// TIA Portal V16 export
// export: Created 2022-03-28T07:44:05.4925085Z, ExportSetting WithDefaults, DisplayName Totally Integrated Automation Portal, DisplayVersion V16 Update 5, DisplayName TIA Portal Version Control Interface, DisplayVersion V16 Update 2, DisplayName TIA Portal Openness, DisplayVersion V16 Update 5, DisplayName STEP 7 Professional, DisplayVersion V16 Update 5, DisplayName STEP 7 Safety, DisplayVersion V16, DisplayName WinCC Professional, DisplayVersion V16 Update 5
FUNCTION "fc_03_Alarms" : Void   // FC3, LAD
{ S7_Optimized_Access := 'TRUE' }
VERSION : 0.1
// stored: AutoNumber false, IsIECCheckEnabled false, SetENOAutomatically false, UDAEnableTagReadback false
   VAR_TEMP   // added for the SCL form of the ladder/FBD networks
      _w1 : Bool;
      _w2 : Bool;
      _w3 : Bool;
   END_VAR
BEGIN

REGION Network 1
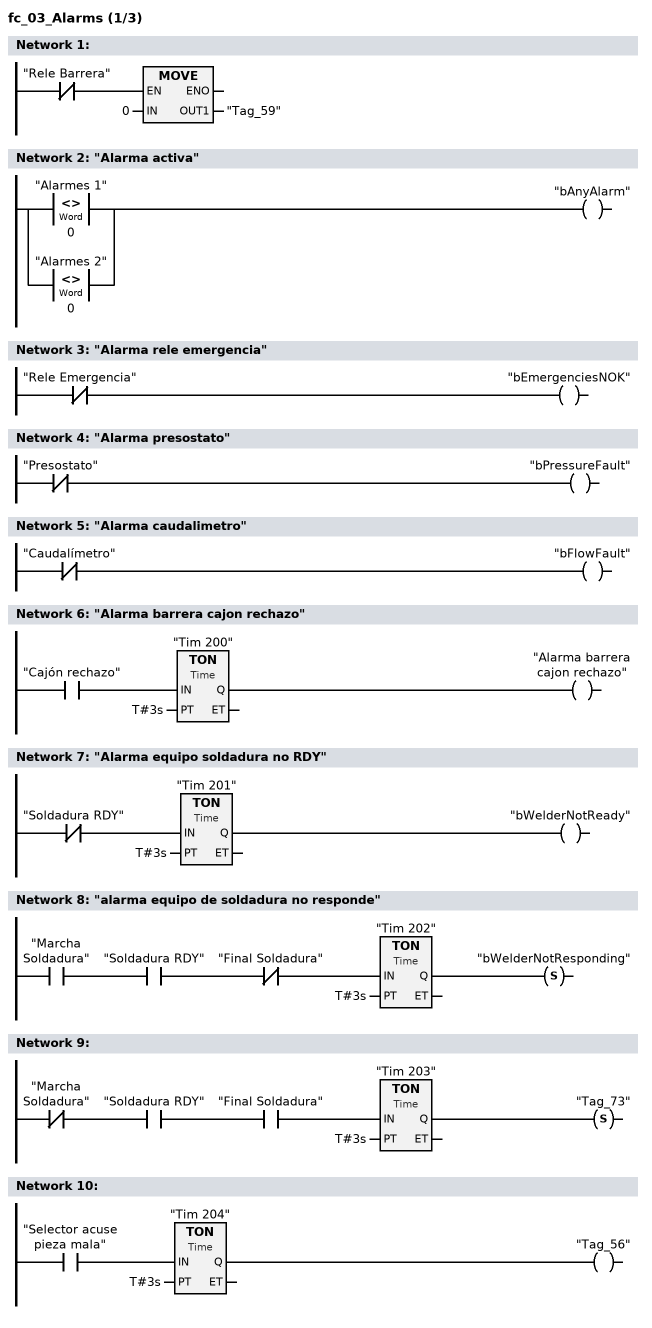
   RUNG wire#powerrail
      I_Contact( "Rele Barrera" )
      Move(in := 0, out1 => "Tag_59")
   END_RUNG
   // the same network as SCL:
   IF NOT "Rele Barrera" THEN "Tag_59" := 0; END_IF;
END_REGION

REGION Network 2: "Alarma activa"
   RUNG wire#powerrail
      { S7_Templates := "SrcType := Word" } NE_Contact(in1 := "Alarmes 1", in2 := 0)
      wire#w1
      Coil( "bAnyAlarm" )
   END_RUNG
   RUNG wire#powerrail
      { S7_Templates := "SrcType := Word" } NE_Contact(in1 := "Alarmes 2", in2 := 0)
   END_RUNG wire#w1
   // the same network as SCL:
   "bAnyAlarm" := ("Alarmes 1" <> 0) OR ("Alarmes 2" <> 0);
END_REGION

REGION Network 3: "Alarma rele emergencia"
   RUNG wire#powerrail
      I_Contact( "Rele Emergencia" )
      Coil( "bEmergenciesNOK" )
   END_RUNG
   // the same network as SCL:
   "bEmergenciesNOK" := NOT "Rele Emergencia";
END_REGION

REGION Network 4: "Alarma presostato"
   RUNG wire#powerrail
      I_Contact( "Presostato" )
      Coil( "bPressureFault" )
   END_RUNG
   // the same network as SCL:
   "bPressureFault" := NOT "Presostato";
END_REGION

REGION Network 5: "Alarma caudalimetro"
   RUNG wire#powerrail
      I_Contact( "Caudalímetro" )
      Coil( "bFlowFault" )
   END_RUNG
   // the same network as SCL:
   "bFlowFault" := NOT "Caudalímetro";
END_REGION

REGION Network 6: "Alarma barrera cajon rechazo"
   RUNG wire#powerrail
      Contact( "Cajón rechazo" )
      { S7_Templates := "time_type := Time" } "Tim 200".TON(pt := T#3s, et =>)
      Coil( "Alarma barrera cajon rechazo" )
   END_RUNG
   // the same network as SCL:
   "Tim 200".TON(IN := "Cajón rechazo", PT := T#3s);
   "Alarma barrera cajon rechazo" := "Tim 200".Q;
END_REGION

REGION Network 7: "Alarma equipo soldadura no RDY"
   RUNG wire#powerrail
      I_Contact( "Soldadura RDY" )
      { S7_Templates := "time_type := Time" } "Tim 201".TON(pt := T#3s, et =>)
      Coil( "bWelderNotReady" )
   END_RUNG
   // the same network as SCL:
   "Tim 201".TON(IN := NOT "Soldadura RDY", PT := T#3s);
   "bWelderNotReady" := "Tim 201".Q;
END_REGION

REGION Network 8: "alarma equipo de soldadura no responde"
   RUNG wire#powerrail
      Contact( "Marcha Soldadura" )
      Contact( "Soldadura RDY" )
      I_Contact( "Final Soldadura" )
      { S7_Templates := "time_type := Time" } "Tim 202".TON(pt := T#3s, et =>)
      S_Coil( "bWelderNotResponding" )
   END_RUNG
   // the same network as SCL:
   "Tim 202".TON(IN := "Marcha Soldadura" AND "Soldadura RDY" AND NOT "Final Soldadura", PT := T#3s);
   IF "Tim 202".Q THEN "bWelderNotResponding" := TRUE; END_IF;
END_REGION

REGION Network 9
   RUNG wire#powerrail
      I_Contact( "Marcha Soldadura" )
      Contact( "Soldadura RDY" )
      Contact( "Final Soldadura" )
      { S7_Templates := "time_type := Time" } "Tim 203".TON(pt := T#3s, et =>)
      S_Coil( "Tag_73" )
   END_RUNG
   // the same network as SCL:
   "Tim 203".TON(IN := NOT "Marcha Soldadura" AND "Soldadura RDY" AND "Final Soldadura", PT := T#3s);
   IF "Tim 203".Q THEN "Tag_73" := TRUE; END_IF;
END_REGION

REGION Network 10
   RUNG wire#powerrail
      Contact( "Selector acuse pieza mala" )
      { S7_Templates := "time_type := Time" } "Tim 204".TON(pt := T#3s, et =>)
      Coil( "Tag_56" )
   END_RUNG
   // the same network as SCL:
   "Tim 204".TON(IN := "Selector acuse pieza mala", PT := T#3s);
   "Tag_56" := "Tim 204".Q;
END_REGION

REGION Network 12: Alarmas Pinza 1
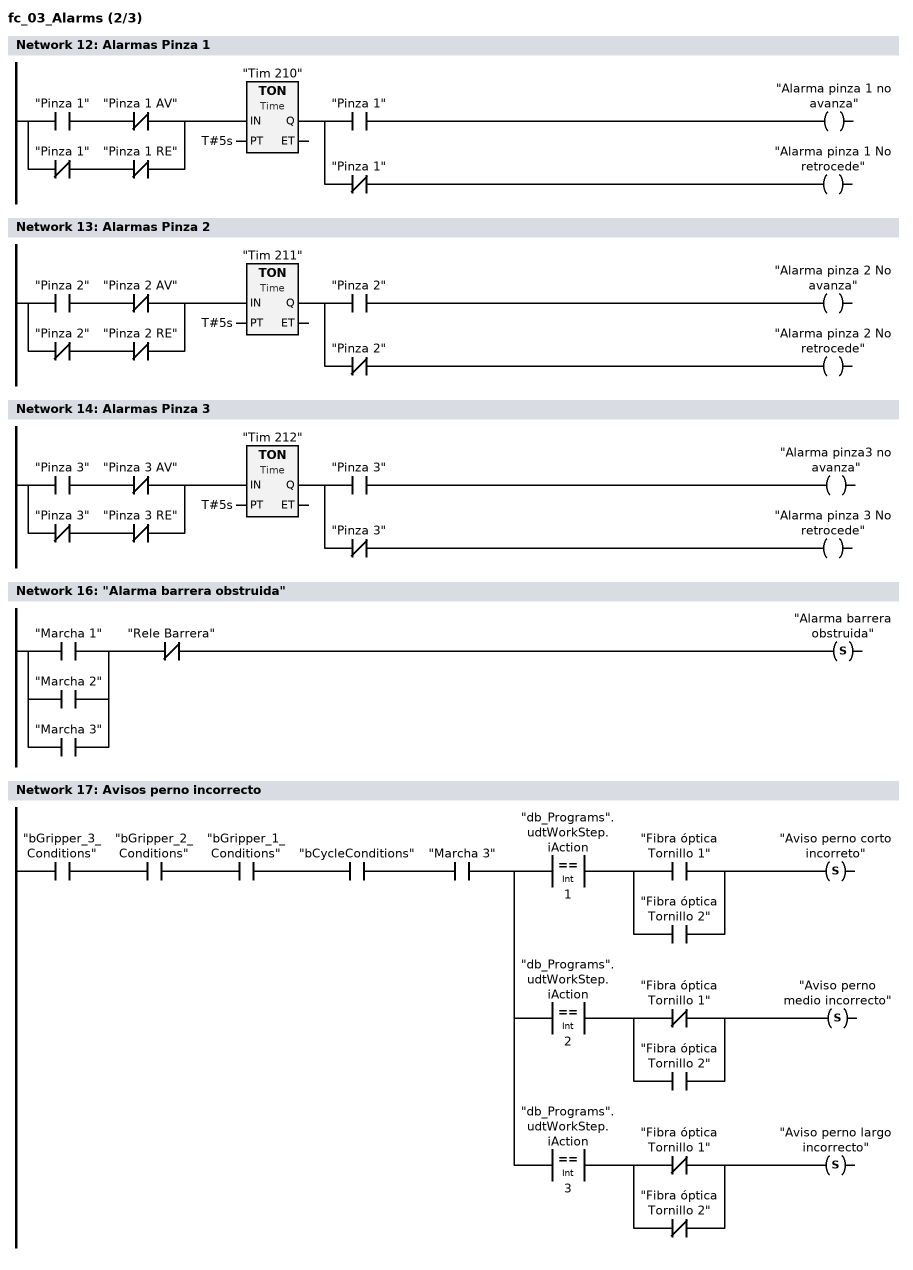
   RUNG wire#powerrail
      Contact( "Pinza 1" )
      I_Contact( "Pinza 1 AV" )
      wire#w1
      { S7_Templates := "time_type := Time" } "Tim 210".TON(pt := T#5s, et =>)
      wire#w2
      Contact( "Pinza 1" )
      Coil( "Alarma pinza 1 no avanza" )
   END_RUNG
   RUNG wire#powerrail
      I_Contact( "Pinza 1" )
      I_Contact( "Pinza 1 RE" )
   END_RUNG wire#w1
   RUNG wire#w2
      I_Contact( "Pinza 1" )
      Coil( "Alarma pinza 1 No retrocede" )
   END_RUNG
   // the same network as SCL:
   "Tim 210".TON(IN := ("Pinza 1" AND NOT "Pinza 1 AV") OR (NOT "Pinza 1" AND NOT "Pinza 1 RE"), PT := T#5s);
   "Alarma pinza 1 no avanza" := "Tim 210".Q AND "Pinza 1";
   "Alarma pinza 1 No retrocede" := "Tim 210".Q AND NOT "Pinza 1";
END_REGION

REGION Network 13: Alarmas Pinza 2
   RUNG wire#powerrail
      Contact( "Pinza 2" )
      I_Contact( "Pinza 2 AV" )
      wire#w1
      { S7_Templates := "time_type := Time" } "Tim 211".TON(pt := T#5s, et =>)
      wire#w2
      Contact( "Pinza 2" )
      Coil( "Alarma pinza 2 No avanza" )
   END_RUNG
   RUNG wire#powerrail
      I_Contact( "Pinza 2" )
      I_Contact( "Pinza 2 RE" )
   END_RUNG wire#w1
   RUNG wire#w2
      I_Contact( "Pinza 2" )
      Coil( "Alarma pinza 2 No retrocede" )
   END_RUNG
   // the same network as SCL:
   "Tim 211".TON(IN := ("Pinza 2" AND NOT "Pinza 2 AV") OR (NOT "Pinza 2" AND NOT "Pinza 2 RE"), PT := T#5s);
   "Alarma pinza 2 No avanza" := "Tim 211".Q AND "Pinza 2";
   "Alarma pinza 2 No retrocede" := "Tim 211".Q AND NOT "Pinza 2";
END_REGION

REGION Network 14: Alarmas Pinza 3
   RUNG wire#powerrail
      Contact( "Pinza 3" )
      I_Contact( "Pinza 3 AV" )
      wire#w1
      { S7_Templates := "time_type := Time" } "Tim 212".TON(pt := T#5s, et =>)
      wire#w2
      Contact( "Pinza 3" )
      Coil( "Alarma pinza3 no avanza" )
   END_RUNG
   RUNG wire#powerrail
      I_Contact( "Pinza 3" )
      I_Contact( "Pinza 3 RE" )
   END_RUNG wire#w1
   RUNG wire#w2
      I_Contact( "Pinza 3" )
      Coil( "Alarma pinza 3 No retrocede" )
   END_RUNG
   // the same network as SCL:
   "Tim 212".TON(IN := ("Pinza 3" AND NOT "Pinza 3 AV") OR (NOT "Pinza 3" AND NOT "Pinza 3 RE"), PT := T#5s);
   "Alarma pinza3 no avanza" := "Tim 212".Q AND "Pinza 3";
   "Alarma pinza 3 No retrocede" := "Tim 212".Q AND NOT "Pinza 3";
END_REGION

REGION Network 16: "Alarma barrera obstruida"
   RUNG wire#powerrail
      Contact( "Marcha 1" )
      wire#w1
      I_Contact( "Rele Barrera" )
      S_Coil( "Alarma barrera obstruida" )
   END_RUNG
   RUNG wire#powerrail
      Contact( "Marcha 2" )
   END_RUNG wire#w1
   RUNG wire#powerrail
      Contact( "Marcha 3" )
   END_RUNG wire#w1
   // the same network as SCL:
   IF ("Marcha 1" OR "Marcha 2" OR "Marcha 3") AND NOT "Rele Barrera" THEN
       "Alarma barrera obstruida" := TRUE;
   END_IF;
END_REGION

REGION Network 17: Avisos perno incorrecto
   RUNG wire#powerrail
      Contact( "bGripper_3_Conditions" )
      Contact( "bGripper_2_Conditions" )
      Contact( "bGripper_1_Conditions" )
      Contact( "bCycleConditions" )
      Contact( "Marcha 3" )
      wire#w1
      { S7_Templates := "SrcType := Int" } EQ_Contact(in1 := "db_Programs".udtWorkStep.iAction, in2 := 1)
      wire#w2
      Contact( "Fibra óptica Tornillo 1" )
      wire#w3
      S_Coil( "Aviso perno corto incorreto" )
   END_RUNG
   RUNG wire#w2
      Contact( "Fibra óptica Tornillo 2" )
   END_RUNG wire#w3
   RUNG wire#w1
      { S7_Templates := "SrcType := Int" } EQ_Contact(in1 := "db_Programs".udtWorkStep.iAction, in2 := 2)
      wire#w4
      I_Contact( "Fibra óptica Tornillo 1" )
      wire#w5
      S_Coil( "Aviso perno medio incorrecto" )
   END_RUNG
   RUNG wire#w4
      Contact( "Fibra óptica Tornillo 2" )
   END_RUNG wire#w5
   RUNG wire#w1
      { S7_Templates := "SrcType := Int" } EQ_Contact(in1 := "db_Programs".udtWorkStep.iAction, in2 := 3)
      wire#w6
      I_Contact( "Fibra óptica Tornillo 1" )
      wire#w7
      S_Coil( "Aviso perno largo incorrecto" )
   END_RUNG
   RUNG wire#w6
      I_Contact( "Fibra óptica Tornillo 2" )
   END_RUNG wire#w7
   // the same network as SCL:
   #_w1 := "bGripper_3_Conditions" AND "bGripper_2_Conditions" AND "bGripper_1_Conditions" AND "bCycleConditions" AND "Marcha 3";
   IF #_w1 AND ("db_Programs".udtWorkStep.iAction = 1) AND ("Fibra óptica Tornillo 1" OR "Fibra óptica Tornillo 2") THEN
       "Aviso perno corto incorreto" := TRUE;
   END_IF;
   IF #_w1 AND ("db_Programs".udtWorkStep.iAction = 2) AND (NOT "Fibra óptica Tornillo 1" OR "Fibra óptica Tornillo 2") THEN
       "Aviso perno medio incorrecto" := TRUE;
   END_IF;
   IF #_w1 AND ("db_Programs".udtWorkStep.iAction = 3) AND (NOT "Fibra óptica Tornillo 1" OR NOT "Fibra óptica Tornillo 2") THEN
       "Aviso perno largo incorrecto" := TRUE;
   END_IF;
END_REGION

REGION Network 18: Avisos perno incorrecto
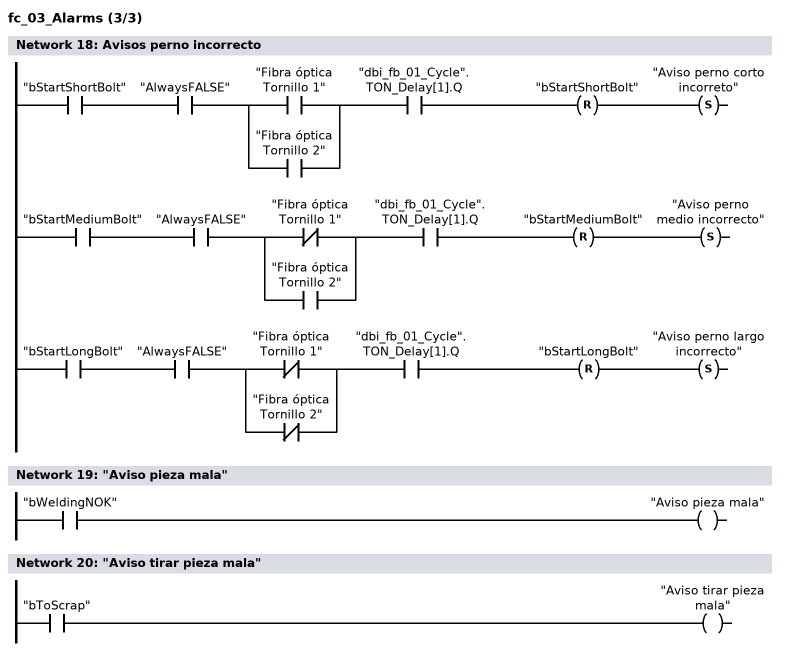
   RUNG wire#powerrail
      Contact( "bStartShortBolt" )
      Contact( "AlwaysFALSE" )
      wire#w1
      Contact( "Fibra óptica Tornillo 1" )
      wire#w2
      Contact( "dbi_fb_01_Cycle".TON_Delay[1].Q )
      R_Coil( "bStartShortBolt" )
      S_Coil( "Aviso perno corto incorreto" )
   END_RUNG
   RUNG wire#w1
      Contact( "Fibra óptica Tornillo 2" )
   END_RUNG wire#w2
   RUNG wire#powerrail
      Contact( "bStartMediumBolt" )
      Contact( "AlwaysFALSE" )
      wire#w3
      I_Contact( "Fibra óptica Tornillo 1" )
      wire#w4
      Contact( "dbi_fb_01_Cycle".TON_Delay[1].Q )
      R_Coil( "bStartMediumBolt" )
      S_Coil( "Aviso perno medio incorrecto" )
   END_RUNG
   RUNG wire#w3
      Contact( "Fibra óptica Tornillo 2" )
   END_RUNG wire#w4
   RUNG wire#powerrail
      Contact( "bStartLongBolt" )
      Contact( "AlwaysFALSE" )
      wire#w5
      I_Contact( "Fibra óptica Tornillo 1" )
      wire#w6
      Contact( "dbi_fb_01_Cycle".TON_Delay[1].Q )
      R_Coil( "bStartLongBolt" )
      S_Coil( "Aviso perno largo incorrecto" )
   END_RUNG
   RUNG wire#w5
      I_Contact( "Fibra óptica Tornillo 2" )
   END_RUNG wire#w6
   // the same network as SCL:
   #_w1 := "bStartShortBolt" AND "AlwaysFALSE" AND ("Fibra óptica Tornillo 1" OR "Fibra óptica Tornillo 2") AND "dbi_fb_01_Cycle".TON_Delay[1].Q;
   IF #_w1 THEN
       "bStartShortBolt" := FALSE;
       "Aviso perno corto incorreto" := TRUE;
   END_IF;
   #_w2 := "bStartMediumBolt" AND "AlwaysFALSE" AND (NOT "Fibra óptica Tornillo 1" OR "Fibra óptica Tornillo 2") AND "dbi_fb_01_Cycle".TON_Delay[1].Q;
   IF #_w2 THEN
       "bStartMediumBolt" := FALSE;
       "Aviso perno medio incorrecto" := TRUE;
   END_IF;
   #_w3 := "bStartLongBolt" AND "AlwaysFALSE" AND (NOT "Fibra óptica Tornillo 1" OR NOT "Fibra óptica Tornillo 2") AND "dbi_fb_01_Cycle".TON_Delay[1].Q;
   IF #_w3 THEN
       "bStartLongBolt" := FALSE;
       "Aviso perno largo incorrecto" := TRUE;
   END_IF;
END_REGION

REGION Network 19: "Aviso pieza mala"
   RUNG wire#powerrail
      Contact( "bWeldingNOK" )
      Coil( "Aviso pieza mala" )
   END_RUNG
   // the same network as SCL:
   "Aviso pieza mala" := "bWeldingNOK";
END_REGION

REGION Network 20: "Aviso tirar pieza mala"
   RUNG wire#powerrail
      Contact( "bToScrap" )
      Coil( "Aviso tirar pieza mala" )
   END_RUNG
   // the same network as SCL:
   "Aviso tirar pieza mala" := "bToScrap";
END_REGION
END_FUNCTION
